REGION Network 1: HS01 / HS02: Contador de veces pulsado sin abrir puerta
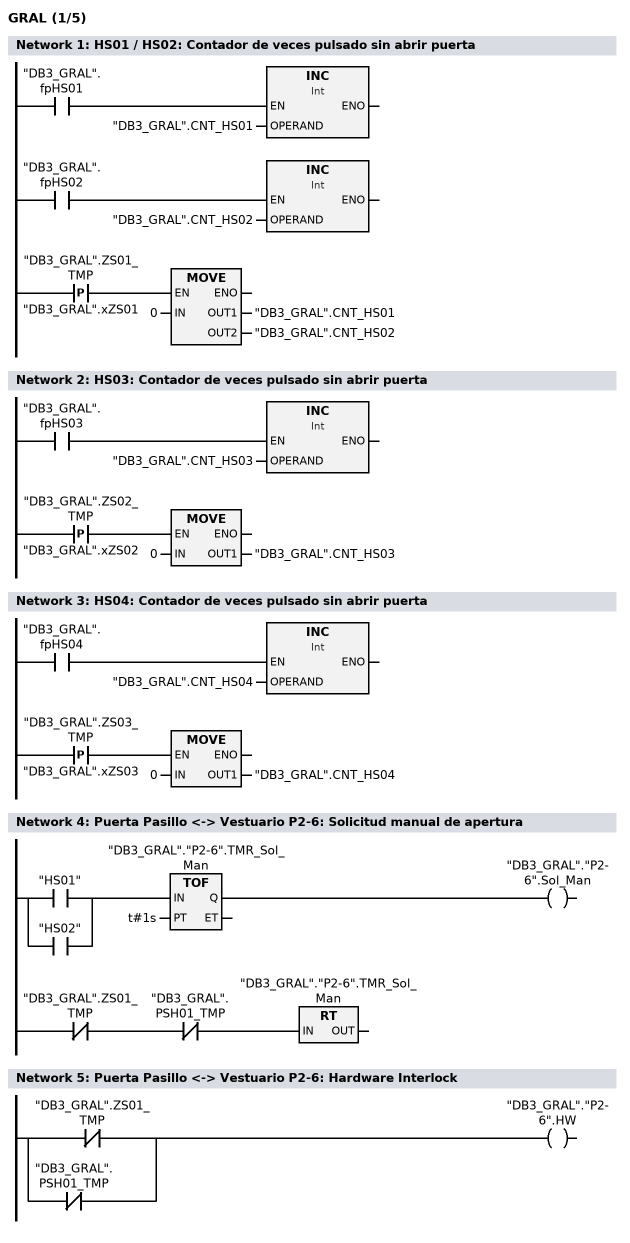
   RUNG wire#powerrail
      Contact( "DB3_GRAL".fpHS01 )
      { S7_Templates := "DestType := Int" } Inc( "DB3_GRAL".CNT_HS01 )
   END_RUNG
   RUNG wire#powerrail
      Contact( "DB3_GRAL".fpHS02 )
      { S7_Templates := "DestType := Int" } Inc( "DB3_GRAL".CNT_HS02 )
   END_RUNG
   RUNG wire#powerrail
      P_Contact(operand := "DB3_GRAL".ZS01_TMP, bit := "DB3_GRAL".xZS01)
      Move(in := 0, out1 => "DB3_GRAL".CNT_HS01, out2 => "DB3_GRAL".CNT_HS02)
   END_RUNG
   // the same network as SCL:
   IF "DB3_GRAL".fpHS01 THEN "DB3_GRAL".CNT_HS01 := "DB3_GRAL".CNT_HS01 + 1; END_IF;
   IF "DB3_GRAL".fpHS02 THEN "DB3_GRAL".CNT_HS02 := "DB3_GRAL".CNT_HS02 + 1; END_IF;
   #_w1 := "DB3_GRAL".ZS01_TMP AND NOT "DB3_GRAL".xZS01;   // rising edge of "DB3_GRAL".ZS01_TMP
   "DB3_GRAL".xZS01 := "DB3_GRAL".ZS01_TMP;
   IF #_w1 THEN
       "DB3_GRAL".CNT_HS01 := 0;
       "DB3_GRAL".CNT_HS02 := 0;
   END_IF;
END_REGION

REGION Network 2: HS03: Contador de veces pulsado sin abrir puerta
   RUNG wire#powerrail
      Contact( "DB3_GRAL".fpHS03 )
      { S7_Templates := "DestType := Int" } Inc( "DB3_GRAL".CNT_HS03 )
   END_RUNG
   RUNG wire#powerrail
      P_Contact(operand := "DB3_GRAL".ZS02_TMP, bit := "DB3_GRAL".xZS02)
      Move(in := 0, out1 => "DB3_GRAL".CNT_HS03)
   END_RUNG
   // the same network as SCL:
   IF "DB3_GRAL".fpHS03 THEN "DB3_GRAL".CNT_HS03 := "DB3_GRAL".CNT_HS03 + 1; END_IF;
   #_w1 := "DB3_GRAL".ZS02_TMP AND NOT "DB3_GRAL".xZS02;   // rising edge of "DB3_GRAL".ZS02_TMP
   "DB3_GRAL".xZS02 := "DB3_GRAL".ZS02_TMP;
   IF #_w1 THEN "DB3_GRAL".CNT_HS03 := 0; END_IF;
END_REGION

REGION Network 3: HS04: Contador de veces pulsado sin abrir puerta
   RUNG wire#powerrail
      Contact( "DB3_GRAL".fpHS04 )
      { S7_Templates := "DestType := Int" } Inc( "DB3_GRAL".CNT_HS04 )
   END_RUNG
   RUNG wire#powerrail
      P_Contact(operand := "DB3_GRAL".ZS03_TMP, bit := "DB3_GRAL".xZS03)
      Move(in := 0, out1 => "DB3_GRAL".CNT_HS04)
   END_RUNG
   // the same network as SCL:
   IF "DB3_GRAL".fpHS04 THEN "DB3_GRAL".CNT_HS04 := "DB3_GRAL".CNT_HS04 + 1; END_IF;
   #_w1 := "DB3_GRAL".ZS03_TMP AND NOT "DB3_GRAL".xZS03;   // rising edge of "DB3_GRAL".ZS03_TMP
   "DB3_GRAL".xZS03 := "DB3_GRAL".ZS03_TMP;
   IF #_w1 THEN "DB3_GRAL".CNT_HS04 := 0; END_IF;
END_REGION

REGION Network 4: Puerta Pasillo <-> Vestuario P2-6: Solicitud manual de apertura
   "DB3_GRAL"."P2-6".TMR_Sol_Man.TOF(IN := "HS01" OR "HS02", PT := t#1s);
   "DB3_GRAL"."P2-6".Sol_Man := "DB3_GRAL"."P2-6".TMR_Sol_Man.Q;
   IF NOT "DB3_GRAL".ZS01_TMP AND NOT "DB3_GRAL".PSH01_TMP THEN
       RESET_TIMER("DB3_GRAL"."P2-6".TMR_Sol_Man);
   END_IF;
END_REGION

REGION Network 5: Puerta Pasillo <-> Vestuario P2-6: Hardware Interlock
   RUNG wire#powerrail
      I_Contact( "DB3_GRAL".ZS01_TMP )
      wire#w1
      Coil( "DB3_GRAL"."P2-6".HW )
   END_RUNG
   RUNG wire#powerrail
      I_Contact( "DB3_GRAL".PSH01_TMP )
   END_RUNG wire#w1
   // the same network as SCL:
   "DB3_GRAL"."P2-6".HW := NOT "DB3_GRAL".ZS01_TMP OR NOT "DB3_GRAL".PSH01_TMP;
END_REGION

REGION Network 6: Puerta Pasillo <-> Vestuario P2-6: Comando apertura
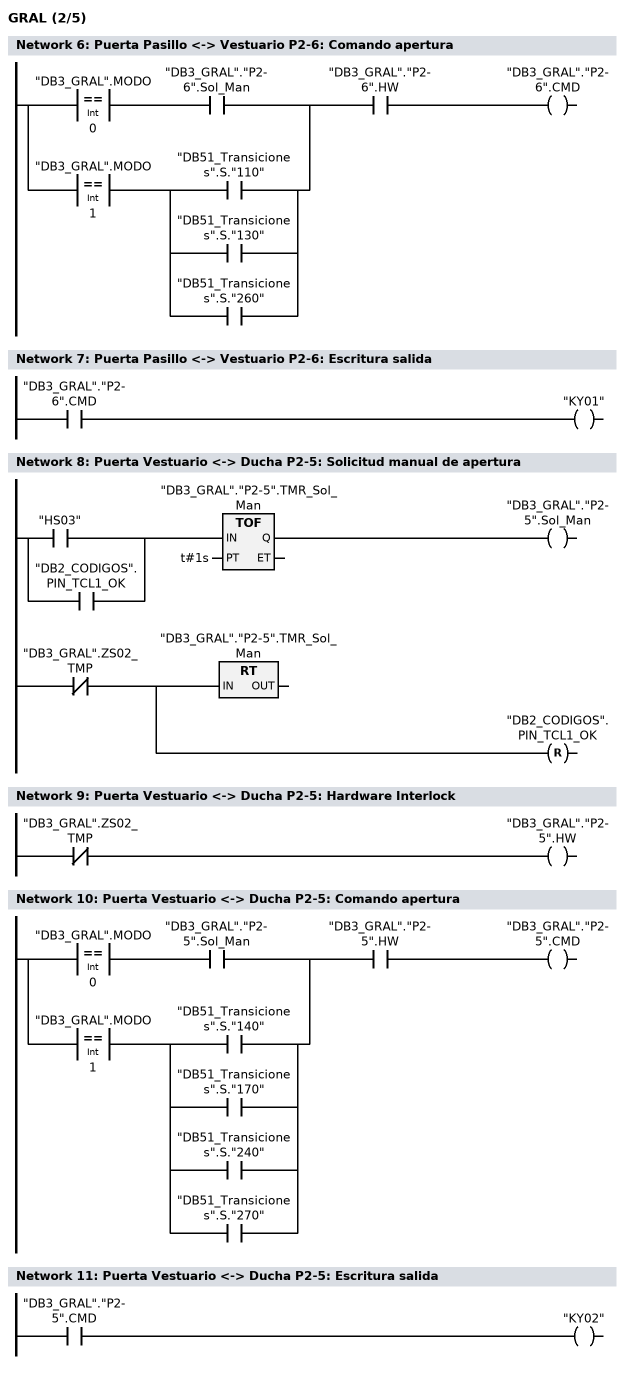
   RUNG wire#powerrail
      { S7_Templates := "SrcType := Int" } EQ_Contact(in1 := "DB3_GRAL".MODO, in2 := 0)
      Contact( "DB3_GRAL"."P2-6".Sol_Man )
      wire#w1
      Contact( "DB3_GRAL"."P2-6".HW )
      Coil( "DB3_GRAL"."P2-6".CMD )
   END_RUNG
   RUNG wire#powerrail
      { S7_Templates := "SrcType := Int" } EQ_Contact(in1 := "DB3_GRAL".MODO, in2 := 1)
      wire#w2
      Contact( "DB51_Transiciones".S."110" )
   END_RUNG wire#w1
   RUNG wire#w2
      Contact( "DB51_Transiciones".S."130" )
   END_RUNG wire#w1
   RUNG wire#w2
      Contact( "DB51_Transiciones".S."260" )
   END_RUNG wire#w1
   // the same network as SCL:
   "DB3_GRAL"."P2-6".CMD := ((("DB3_GRAL".MODO = 0) AND "DB3_GRAL"."P2-6".Sol_Man) OR (("DB3_GRAL".MODO = 1) AND ("DB51_Transiciones".S."110" OR "DB51_Transiciones".S."130" OR "DB51_Transiciones".S."260"))) AND "DB3_GRAL"."P2-6".HW;
END_REGION

REGION Network 7: Puerta Pasillo <-> Vestuario P2-6: Escritura salida
   RUNG wire#powerrail
      Contact( "DB3_GRAL"."P2-6".CMD )
      Coil( "KY01" )
   END_RUNG
   // the same network as SCL:
   "KY01" := "DB3_GRAL"."P2-6".CMD;
END_REGION

REGION Network 8: Puerta Vestuario <-> Ducha P2-5: Solicitud manual de apertura
   "DB3_GRAL"."P2-5".TMR_Sol_Man.TOF(IN := "HS03" OR "DB2_CODIGOS".PIN_TCL1_OK, PT := t#1s);
   "DB3_GRAL"."P2-5".Sol_Man := "DB3_GRAL"."P2-5".TMR_Sol_Man.Q;
   IF NOT "DB3_GRAL".ZS02_TMP THEN
       RESET_TIMER("DB3_GRAL"."P2-5".TMR_Sol_Man);
       "DB2_CODIGOS".PIN_TCL1_OK := FALSE;
   END_IF;
END_REGION

REGION Network 9: Puerta Vestuario <-> Ducha P2-5: Hardware Interlock
   RUNG wire#powerrail
      I_Contact( "DB3_GRAL".ZS02_TMP )
      Coil( "DB3_GRAL"."P2-5".HW )
   END_RUNG
   // the same network as SCL:
   "DB3_GRAL"."P2-5".HW := NOT "DB3_GRAL".ZS02_TMP;
END_REGION

REGION Network 10: Puerta Vestuario <-> Ducha P2-5: Comando apertura
   RUNG wire#powerrail
      { S7_Templates := "SrcType := Int" } EQ_Contact(in1 := "DB3_GRAL".MODO, in2 := 0)
      Contact( "DB3_GRAL"."P2-5".Sol_Man )
      wire#w1
      Contact( "DB3_GRAL"."P2-5".HW )
      Coil( "DB3_GRAL"."P2-5".CMD )
   END_RUNG
   RUNG wire#powerrail
      { S7_Templates := "SrcType := Int" } EQ_Contact(in1 := "DB3_GRAL".MODO, in2 := 1)
      wire#w2
      Contact( "DB51_Transiciones".S."140" )
   END_RUNG wire#w1
   RUNG wire#w2
      Contact( "DB51_Transiciones".S."170" )
   END_RUNG wire#w1
   RUNG wire#w2
      Contact( "DB51_Transiciones".S."240" )
   END_RUNG wire#w1
   RUNG wire#w2
      Contact( "DB51_Transiciones".S."270" )
   END_RUNG wire#w1
   // the same network as SCL:
   "DB3_GRAL"."P2-5".CMD := ((("DB3_GRAL".MODO = 0) AND "DB3_GRAL"."P2-5".Sol_Man) OR (("DB3_GRAL".MODO = 1) AND ("DB51_Transiciones".S."140" OR "DB51_Transiciones".S."170" OR "DB51_Transiciones".S."240" OR "DB51_Transiciones".S."270"))) AND "DB3_GRAL"."P2-5".HW;
END_REGION

REGION Network 11: Puerta Vestuario <-> Ducha P2-5: Escritura salida
   RUNG wire#powerrail
      Contact( "DB3_GRAL"."P2-5".CMD )
      Coil( "KY02" )
   END_RUNG
   // the same network as SCL:
   "KY02" := "DB3_GRAL"."P2-5".CMD;
END_REGION

REGION Network 12: Puerta Ducha <-> Bioterio P2-4: Solicitud manual de apertura
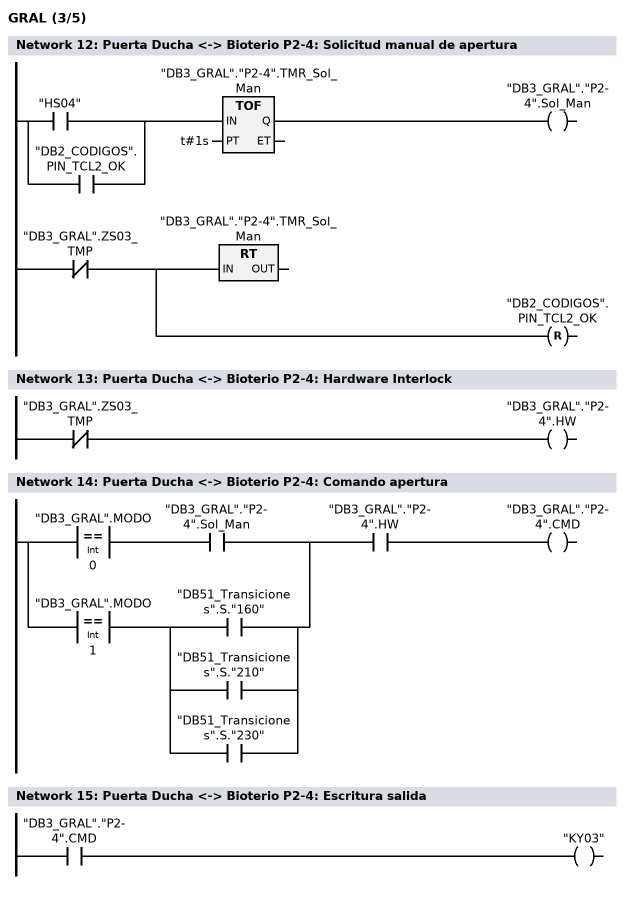
   "DB3_GRAL"."P2-4".TMR_Sol_Man.TOF(IN := "HS04" OR "DB2_CODIGOS".PIN_TCL2_OK, PT := t#1s);
   "DB3_GRAL"."P2-4".Sol_Man := "DB3_GRAL"."P2-4".TMR_Sol_Man.Q;
   IF NOT "DB3_GRAL".ZS03_TMP THEN
       RESET_TIMER("DB3_GRAL"."P2-4".TMR_Sol_Man);
       "DB2_CODIGOS".PIN_TCL2_OK := FALSE;
   END_IF;
END_REGION

REGION Network 13: Puerta Ducha <-> Bioterio P2-4: Hardware Interlock
   RUNG wire#powerrail
      I_Contact( "DB3_GRAL".ZS03_TMP )
      Coil( "DB3_GRAL"."P2-4".HW )
   END_RUNG
   // the same network as SCL:
   "DB3_GRAL"."P2-4".HW := NOT "DB3_GRAL".ZS03_TMP;
END_REGION

REGION Network 14: Puerta Ducha <-> Bioterio P2-4: Comando apertura
   RUNG wire#powerrail
      { S7_Templates := "SrcType := Int" } EQ_Contact(in1 := "DB3_GRAL".MODO, in2 := 0)
      Contact( "DB3_GRAL"."P2-4".Sol_Man )
      wire#w1
      Contact( "DB3_GRAL"."P2-4".HW )
      Coil( "DB3_GRAL"."P2-4".CMD )
   END_RUNG
   RUNG wire#powerrail
      { S7_Templates := "SrcType := Int" } EQ_Contact(in1 := "DB3_GRAL".MODO, in2 := 1)
      wire#w2
      Contact( "DB51_Transiciones".S."160" )
   END_RUNG wire#w1
   RUNG wire#w2
      Contact( "DB51_Transiciones".S."210" )
   END_RUNG wire#w1
   RUNG wire#w2
      Contact( "DB51_Transiciones".S."230" )
   END_RUNG wire#w1
   // the same network as SCL:
   "DB3_GRAL"."P2-4".CMD := ((("DB3_GRAL".MODO = 0) AND "DB3_GRAL"."P2-4".Sol_Man) OR (("DB3_GRAL".MODO = 1) AND ("DB51_Transiciones".S."160" OR "DB51_Transiciones".S."210" OR "DB51_Transiciones".S."230"))) AND "DB3_GRAL"."P2-4".HW;
END_REGION

REGION Network 15: Puerta Ducha <-> Bioterio P2-4: Escritura salida
   RUNG wire#powerrail
      Contact( "DB3_GRAL"."P2-4".CMD )
      Coil( "KY03" )
   END_RUNG
   // the same network as SCL:
   "KY03" := "DB3_GRAL"."P2-4".CMD;
END_REGION

REGION Network 16: Ducha - Electroválvula: Solicitud manual de apertura
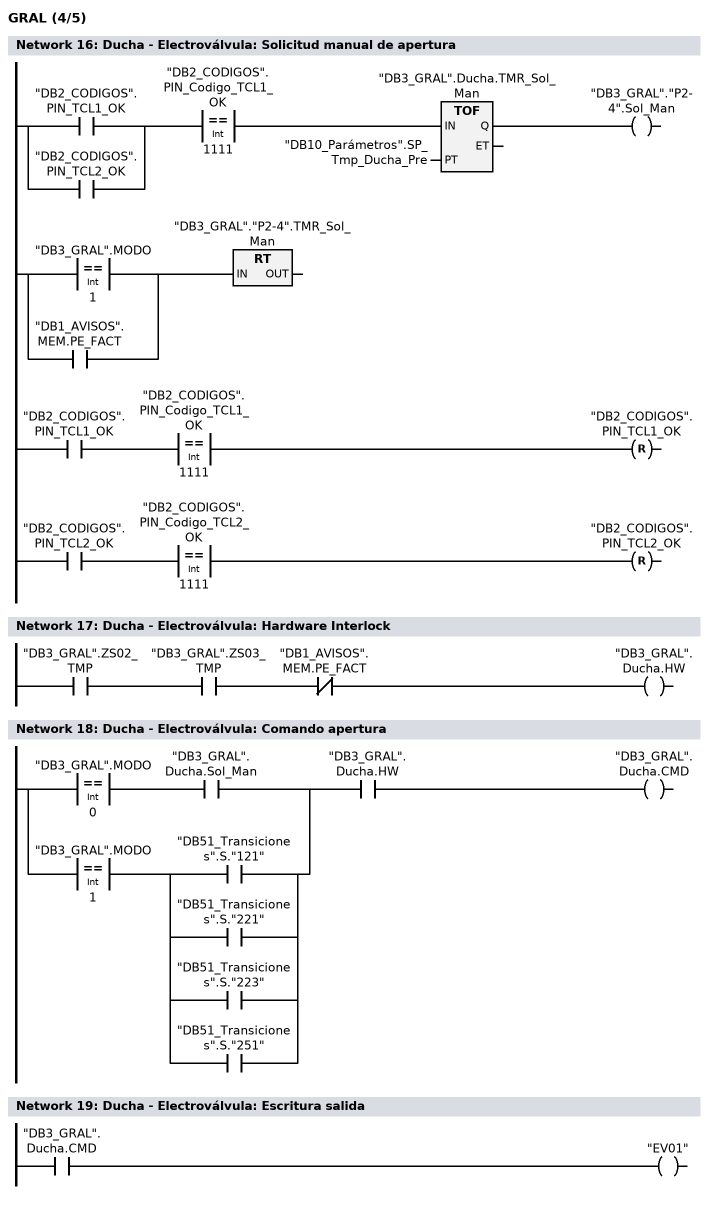
   "DB3_GRAL".Ducha.TMR_Sol_Man.TOF(IN := ("DB2_CODIGOS".PIN_TCL1_OK OR "DB2_CODIGOS".PIN_TCL2_OK) AND ("DB2_CODIGOS".PIN_Codigo_TCL1_OK = 1111),
                           PT := "DB10_Parámetros".SP_Tmp_Ducha_Pre);
   "DB3_GRAL"."P2-4".Sol_Man := "DB3_GRAL".Ducha.TMR_Sol_Man.Q;
   IF ("DB3_GRAL".MODO = 1) OR "DB1_AVISOS".MEM.PE_FACT THEN
       RESET_TIMER("DB3_GRAL"."P2-4".TMR_Sol_Man);
   END_IF;
   IF "DB2_CODIGOS".PIN_TCL1_OK AND ("DB2_CODIGOS".PIN_Codigo_TCL1_OK = 1111) THEN
       "DB2_CODIGOS".PIN_TCL1_OK := FALSE;
   END_IF;
   IF "DB2_CODIGOS".PIN_TCL2_OK AND ("DB2_CODIGOS".PIN_Codigo_TCL2_OK = 1111) THEN
       "DB2_CODIGOS".PIN_TCL2_OK := FALSE;
   END_IF;
END_REGION

REGION Network 17: Ducha - Electroválvula: Hardware Interlock
   RUNG wire#powerrail
      Contact( "DB3_GRAL".ZS02_TMP )
      Contact( "DB3_GRAL".ZS03_TMP )
      I_Contact( "DB1_AVISOS".MEM.PE_FACT )
      Coil( "DB3_GRAL".Ducha.HW )
   END_RUNG
   // the same network as SCL:
   "DB3_GRAL".Ducha.HW := "DB3_GRAL".ZS02_TMP AND "DB3_GRAL".ZS03_TMP AND NOT "DB1_AVISOS".MEM.PE_FACT;
END_REGION

REGION Network 18: Ducha - Electroválvula: Comando apertura
   RUNG wire#powerrail
      { S7_Templates := "SrcType := Int" } EQ_Contact(in1 := "DB3_GRAL".MODO, in2 := 0)
      Contact( "DB3_GRAL".Ducha.Sol_Man )
      wire#w1
      Contact( "DB3_GRAL".Ducha.HW )
      Coil( "DB3_GRAL".Ducha.CMD )
   END_RUNG
   RUNG wire#powerrail
      { S7_Templates := "SrcType := Int" } EQ_Contact(in1 := "DB3_GRAL".MODO, in2 := 1)
      wire#w2
      Contact( "DB51_Transiciones".S."121" )
   END_RUNG wire#w1
   RUNG wire#w2
      Contact( "DB51_Transiciones".S."221" )
   END_RUNG wire#w1
   RUNG wire#w2
      Contact( "DB51_Transiciones".S."223" )
   END_RUNG wire#w1
   RUNG wire#w2
      Contact( "DB51_Transiciones".S."251" )
   END_RUNG wire#w1
   // the same network as SCL:
   "DB3_GRAL".Ducha.CMD := ((("DB3_GRAL".MODO = 0) AND "DB3_GRAL".Ducha.Sol_Man) OR (("DB3_GRAL".MODO = 1) AND ("DB51_Transiciones".S."121" OR "DB51_Transiciones".S."221" OR "DB51_Transiciones".S."223" OR "DB51_Transiciones".S."251"))) AND "DB3_GRAL".Ducha.HW;
END_REGION

REGION Network 19: Ducha - Electroválvula: Escritura salida
   RUNG wire#powerrail
      Contact( "DB3_GRAL".Ducha.CMD )
      Coil( "EV01" )
   END_RUNG
   // the same network as SCL:
   "EV01" := "DB3_GRAL".Ducha.CMD;
END_REGION

REGION Network 20: *****************************************************
END_REGION

REGION Network 21: Contador de personas que ingresaron al bioterio
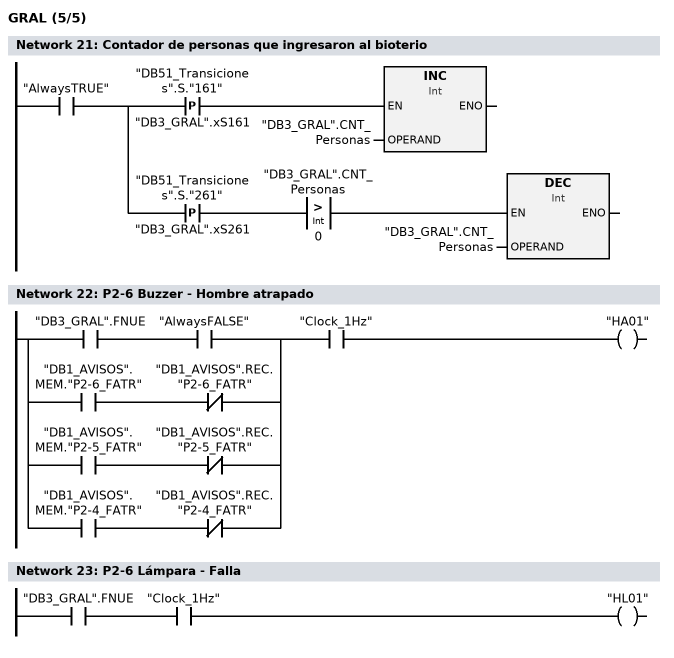
   RUNG wire#powerrail
      Contact( "AlwaysTRUE" )
      wire#w1
      P_Contact(operand := "DB51_Transiciones".S."161", bit := "DB3_GRAL".xS161)
      { S7_Templates := "DestType := Int" } Inc( "DB3_GRAL".CNT_Personas )
   END_RUNG
   RUNG wire#w1
      P_Contact(operand := "DB51_Transiciones".S."261", bit := "DB3_GRAL".xS261)
      { S7_Templates := "SrcType := Int" } GT_Contact(in1 := "DB3_GRAL".CNT_Personas, in2 := 0)
      { S7_Templates := "DestType := Int" } Dec( "DB3_GRAL".CNT_Personas )
   END_RUNG
   // the same network as SCL:
   #_w1 := "AlwaysTRUE" AND "DB51_Transiciones".S."161" AND NOT "DB3_GRAL".xS161;   // rising edge of "DB51_Transiciones".S."161"
   "DB3_GRAL".xS161 := "DB51_Transiciones".S."161";
   IF #_w1 THEN "DB3_GRAL".CNT_Personas := "DB3_GRAL".CNT_Personas + 1; END_IF;
   #_w2 := "AlwaysTRUE" AND "DB51_Transiciones".S."261" AND NOT "DB3_GRAL".xS261;   // rising edge of "DB51_Transiciones".S."261"
   "DB3_GRAL".xS261 := "DB51_Transiciones".S."261";
   IF #_w2 AND ("DB3_GRAL".CNT_Personas > 0) THEN
       "DB3_GRAL".CNT_Personas := "DB3_GRAL".CNT_Personas - 1;
   END_IF;
END_REGION

REGION Network 22: P2-6 Buzzer - Hombre atrapado
   RUNG wire#powerrail
      Contact( "DB3_GRAL".FNUE )
      Contact( "AlwaysFALSE" )
      wire#w1
      Contact( "Clock_1Hz" )
      Coil( "HA01" )
   END_RUNG
   RUNG wire#powerrail
      Contact( "DB1_AVISOS".MEM."P2-6_FATR" )
      I_Contact( "DB1_AVISOS".REC."P2-6_FATR" )
   END_RUNG wire#w1
   RUNG wire#powerrail
      Contact( "DB1_AVISOS".MEM."P2-5_FATR" )
      I_Contact( "DB1_AVISOS".REC."P2-5_FATR" )
   END_RUNG wire#w1
   RUNG wire#powerrail
      Contact( "DB1_AVISOS".MEM."P2-4_FATR" )
      I_Contact( "DB1_AVISOS".REC."P2-4_FATR" )
   END_RUNG wire#w1
   // the same network as SCL:
   "HA01" := (("DB3_GRAL".FNUE AND "AlwaysFALSE") OR ("DB1_AVISOS".MEM."P2-6_FATR" AND NOT "DB1_AVISOS".REC."P2-6_FATR") OR ("DB1_AVISOS".MEM."P2-5_FATR" AND NOT "DB1_AVISOS".REC."P2-5_FATR") OR ("DB1_AVISOS".MEM."P2-4_FATR" AND NOT "DB1_AVISOS".REC."P2-4_FATR")) AND "Clock_1Hz";
END_REGION

REGION Network 23: P2-6 Lámpara - Falla
   RUNG wire#powerrail
      Contact( "DB3_GRAL".FNUE )
      Contact( "Clock_1Hz" )
      Coil( "HL01" )
   END_RUNG
   // the same network as SCL:
   "HL01" := "DB3_GRAL".FNUE AND "Clock_1Hz";
END_REGION
END_FUNCTION

FUNCTION "INICIA" : Void   // FC5, LAD
TITLE = Inicialización de datos
{ S7_Optimized_Access := 'TRUE' }
AUTHOR : IGLP
VERSION : 0.1
BEGIN

REGION Network 1: Contacto Magnético P2-6 - Temporizado
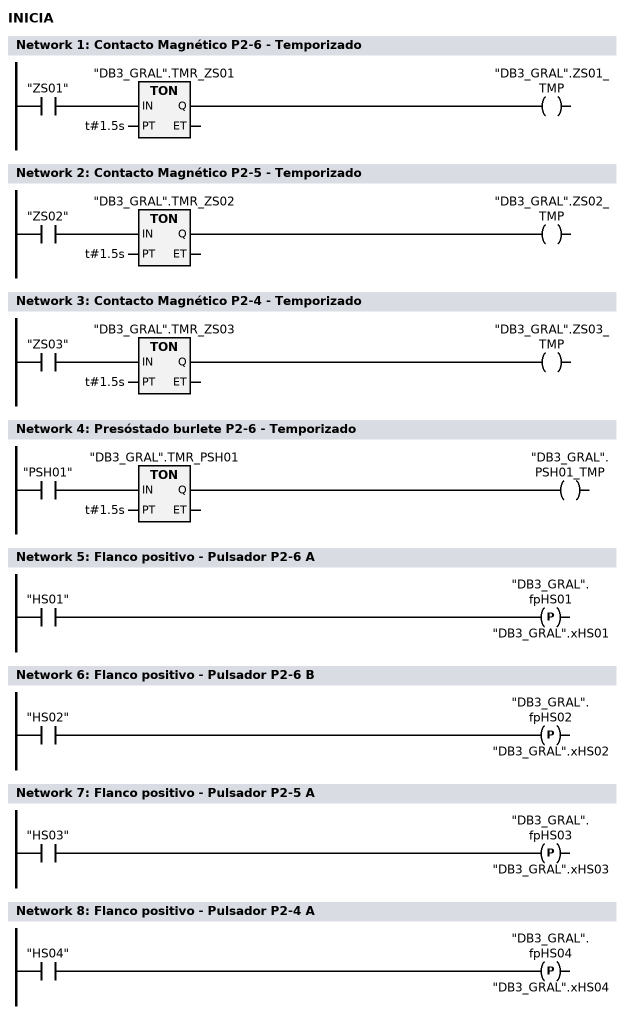
   "DB3_GRAL".TMR_ZS01.TON(IN := "ZS01", PT := t#1.5s);
   "DB3_GRAL".ZS01_TMP := "DB3_GRAL".TMR_ZS01.Q;
END_REGION

REGION Network 2: Contacto Magnético P2-5 - Temporizado
   "DB3_GRAL".TMR_ZS02.TON(IN := "ZS02", PT := t#1.5s);
   "DB3_GRAL".ZS02_TMP := "DB3_GRAL".TMR_ZS02.Q;
END_REGION

REGION Network 3: Contacto Magnético P2-4 - Temporizado
   "DB3_GRAL".TMR_ZS03.TON(IN := "ZS03", PT := t#1.5s);
   "DB3_GRAL".ZS03_TMP := "DB3_GRAL".TMR_ZS03.Q;
END_REGION

REGION Network 4: Presóstado burlete P2-6 - Temporizado
   "DB3_GRAL".TMR_PSH01.TON(IN := "PSH01", PT := t#1.5s);
   "DB3_GRAL".PSH01_TMP := "DB3_GRAL".TMR_PSH01.Q;
END_REGION

REGION Network 5: Flanco positivo - Pulsador P2-6 A
   "DB3_GRAL".fpHS01 := "HS01" AND NOT "DB3_GRAL".xHS01;   // rising edge
   "DB3_GRAL".xHS01 := "HS01";
END_REGION

REGION Network 6: Flanco positivo - Pulsador P2-6 B
   "DB3_GRAL".fpHS02 := "HS02" AND NOT "DB3_GRAL".xHS02;   // rising edge
   "DB3_GRAL".xHS02 := "HS02";
END_REGION

REGION Network 7: Flanco positivo - Pulsador P2-5 A
   "DB3_GRAL".fpHS03 := "HS03" AND NOT "DB3_GRAL".xHS03;   // rising edge
   "DB3_GRAL".xHS03 := "HS03";
END_REGION

REGION Network 8: Flanco positivo - Pulsador P2-4 A
   "DB3_GRAL".fpHS04 := "HS04" AND NOT "DB3_GRAL".xHS04;   // rising edge
   "DB3_GRAL".xHS04 := "HS04";
END_REGION
END_FUNCTION

FUNCTION "AVISOS" : Void   // FC6, LAD
TITLE = Avisos
{ S7_Optimized_Access := 'TRUE' }
AUTHOR : IGLP
VERSION : 0.1
BEGIN

REGION Network 1: Falla: Emergencia actuada
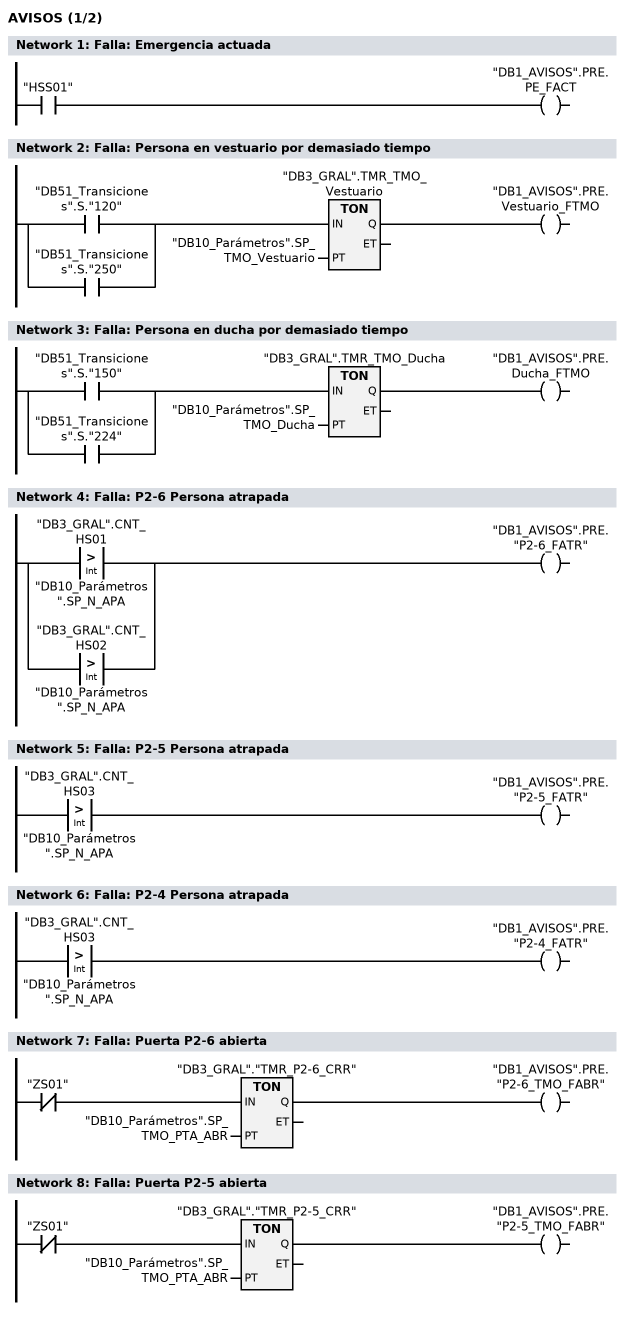
   RUNG wire#powerrail
      Contact( "HSS01" )
      Coil( "DB1_AVISOS".PRE.PE_FACT )
   END_RUNG
   // the same network as SCL:
   "DB1_AVISOS".PRE.PE_FACT := "HSS01";
END_REGION

REGION Network 2: Falla: Persona en vestuario por demasiado tiempo
   "DB3_GRAL".TMR_TMO_Vestuario.TON(IN := "DB51_Transiciones".S."120" OR "DB51_Transiciones".S."250",
                           PT := "DB10_Parámetros".SP_TMO_Vestuario);
   "DB1_AVISOS".PRE.Vestuario_FTMO := "DB3_GRAL".TMR_TMO_Vestuario.Q;
END_REGION

REGION Network 3: Falla: Persona en ducha por demasiado tiempo
   "DB3_GRAL".TMR_TMO_Ducha.TON(IN := "DB51_Transiciones".S."150" OR "DB51_Transiciones".S."224",
                           PT := "DB10_Parámetros".SP_TMO_Ducha);
   "DB1_AVISOS".PRE.Ducha_FTMO := "DB3_GRAL".TMR_TMO_Ducha.Q;
END_REGION

REGION Network 4: Falla: P2-6 Persona atrapada
   RUNG wire#powerrail
      { S7_Templates := "SrcType := Int" } GT_Contact(in1 := "DB3_GRAL".CNT_HS01, in2 := "DB10_Parámetros".SP_N_APA)
      wire#w1
      Coil( "DB1_AVISOS".PRE."P2-6_FATR" )
   END_RUNG
   RUNG wire#powerrail
      { S7_Templates := "SrcType := Int" } GT_Contact(in1 := "DB3_GRAL".CNT_HS02, in2 := "DB10_Parámetros".SP_N_APA)
   END_RUNG wire#w1
   // the same network as SCL:
   "DB1_AVISOS".PRE."P2-6_FATR" := ("DB3_GRAL".CNT_HS01 > "DB10_Parámetros".SP_N_APA) OR ("DB3_GRAL".CNT_HS02 > "DB10_Parámetros".SP_N_APA);
END_REGION

REGION Network 5: Falla: P2-5 Persona atrapada
   RUNG wire#powerrail
      { S7_Templates := "SrcType := Int" } GT_Contact(in1 := "DB3_GRAL".CNT_HS03, in2 := "DB10_Parámetros".SP_N_APA)
      Coil( "DB1_AVISOS".PRE."P2-5_FATR" )
   END_RUNG
   // the same network as SCL:
   "DB1_AVISOS".PRE."P2-5_FATR" := "DB3_GRAL".CNT_HS03 > "DB10_Parámetros".SP_N_APA;
END_REGION

REGION Network 6: Falla: P2-4 Persona atrapada
   RUNG wire#powerrail
      { S7_Templates := "SrcType := Int" } GT_Contact(in1 := "DB3_GRAL".CNT_HS03, in2 := "DB10_Parámetros".SP_N_APA)
      Coil( "DB1_AVISOS".PRE."P2-4_FATR" )
   END_RUNG
   // the same network as SCL:
   "DB1_AVISOS".PRE."P2-4_FATR" := "DB3_GRAL".CNT_HS03 > "DB10_Parámetros".SP_N_APA;
END_REGION

REGION Network 7: Falla: Puerta P2-6 abierta
   "DB3_GRAL"."TMR_P2-6_CRR".TON(IN := NOT "ZS01", PT := "DB10_Parámetros".SP_TMO_PTA_ABR);
   "DB1_AVISOS".PRE."P2-6_TMO_FABR" := "DB3_GRAL"."TMR_P2-6_CRR".Q;
END_REGION

REGION Network 8: Falla: Puerta P2-5 abierta
   "DB3_GRAL"."TMR_P2-5_CRR".TON(IN := NOT "ZS01", PT := "DB10_Parámetros".SP_TMO_PTA_ABR);
   "DB1_AVISOS".PRE."P2-5_TMO_FABR" := "DB3_GRAL"."TMR_P2-5_CRR".Q;
END_REGION

REGION Network 9: Falla: Puerta P2-4 abierta
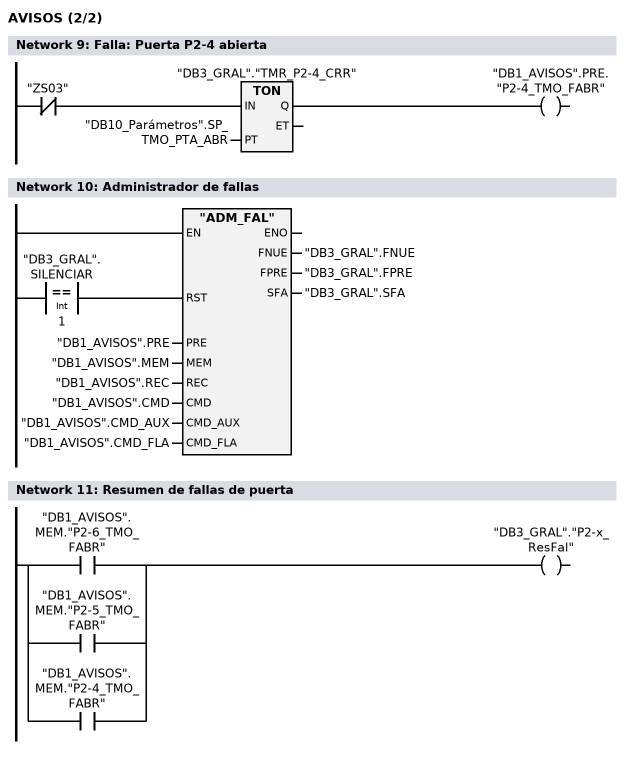
   "DB3_GRAL"."TMR_P2-4_CRR".TON(IN := NOT "ZS03", PT := "DB10_Parámetros".SP_TMO_PTA_ABR);
   "DB1_AVISOS".PRE."P2-4_TMO_FABR" := "DB3_GRAL"."TMR_P2-4_CRR".Q;
END_REGION

REGION Network 10: Administrador de fallas
   RUNG wire#powerrail
      "ADM_FAL"(RST := wire#w1, PRE := "DB1_AVISOS".PRE, MEM := "DB1_AVISOS".MEM, REC := "DB1_AVISOS".REC, CMD := "DB1_AVISOS".CMD, CMD_AUX := "DB1_AVISOS".CMD_AUX, CMD_FLA := "DB1_AVISOS".CMD_FLA, FNUE => "DB3_GRAL".FNUE, FPRE => "DB3_GRAL".FPRE, SFA => "DB3_GRAL".SFA)
   END_RUNG
   RUNG wire#powerrail
      { S7_Templates := "SrcType := Int" } EQ_Contact(in1 := "DB3_GRAL".SILENCIAR, in2 := 1)
   END_RUNG wire#w1
   // the same network as SCL:
   "ADM_FAL"(RST := "DB3_GRAL".SILENCIAR = 1,
             PRE := "DB1_AVISOS".PRE,
             MEM := "DB1_AVISOS".MEM,
             REC := "DB1_AVISOS".REC,
             CMD := "DB1_AVISOS".CMD,
             CMD_AUX := "DB1_AVISOS".CMD_AUX,
             CMD_FLA := "DB1_AVISOS".CMD_FLA,
             FNUE => "DB3_GRAL".FNUE,
             FPRE => "DB3_GRAL".FPRE,
             SFA => "DB3_GRAL".SFA);
END_REGION

REGION Network 11: Resumen de fallas de puerta
   RUNG wire#powerrail
      Contact( "DB1_AVISOS".MEM."P2-6_TMO_FABR" )
      wire#w1
      Coil( "DB3_GRAL"."P2-x_ResFal" )
   END_RUNG
   RUNG wire#powerrail
      Contact( "DB1_AVISOS".MEM."P2-5_TMO_FABR" )
   END_RUNG wire#w1
   RUNG wire#powerrail
      Contact( "DB1_AVISOS".MEM."P2-4_TMO_FABR" )
   END_RUNG wire#w1
   // the same network as SCL:
   "DB3_GRAL"."P2-x_ResFal" := "DB1_AVISOS".MEM."P2-6_TMO_FABR" OR "DB1_AVISOS".MEM."P2-5_TMO_FABR" OR "DB1_AVISOS".MEM."P2-4_TMO_FABR";
END_REGION
END_FUNCTION

FUNCTION "ADM_FAL" : Void   // FC7, LAD
TITLE = Procesador de fallas
{ S7_Optimized_Access := 'FALSE' }
VERSION : 0.1
   VAR_INPUT
      RST : Bool;
   END_VAR
   VAR_OUTPUT
      FNUE : Bool;
      FPRE : Bool;
      SFA : Bool;
   END_VAR
   VAR_IN_OUT
      PRE : "FALLAS";
      aPRE AT PRE : Array[1..2] of Byte;
      MEM : "FALLAS";
      aMEM AT MEM : Array[1..2] of Byte;
      REC : "FALLAS";
      aREC AT REC : Array[1..2] of Byte;
      CMD : "FALLAS";
      aCMD AT CMD : Array[1..2] of Byte;
      CMD_AUX : "FALLAS";
      aCMD_AUX AT CMD_AUX : Array[1..2] of Byte;
      CMD_FLA : "FALLAS";
      aCMD_FLA AT CMD_FLA : Array[1..2] of Byte;
   END_VAR
   VAR_TEMP
      INDICE : Int;
      AUX_FLA_CMD_REC : Byte;
      AUX_Reconocida1 : Byte;
      AUX_Reconocida2 : Byte;
   END_VAR
BEGIN

REGION Network 1: Inicializo
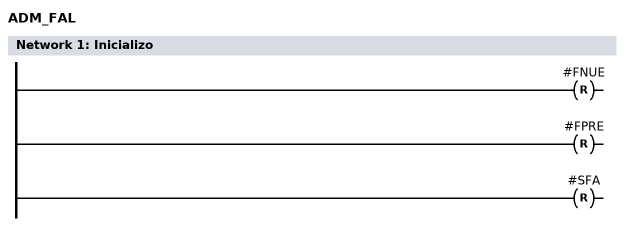
   RUNG wire#powerrail
      R_Coil( #FNUE )
   END_RUNG
   RUNG wire#powerrail
      R_Coil( #FPRE )
   END_RUNG
   RUNG wire#powerrail
      R_Coil( #SFA )
   END_RUNG
   // the same network as SCL:
   #FNUE := FALSE;
   #FPRE := FALSE;
   #SFA := FALSE;
END_REGION

REGION Network 2 (SCL): Comandos reconocimiento: Detección de flancos
   FOR #INDICE := 1 TO 2 DO
       #aCMD_FLA[#INDICE] := (#aCMD[#INDICE] XOR #aCMD_AUX[#INDICE]);
       #aCMD_AUX[#INDICE] := #aCMD[#INDICE];
   END_FOR;
END_REGION

REGION Network 3 (SCL): Memorizo alarmas y reconozco cuando llega flanco
   // Sobre las alarmas reconocidas hay dos operaciones:
   // Set =   (NO(Alarma Presente) * NO(Alarma Memorizada))  + (Alarma Memorizada * Flanco Cmd. Reconocimiento)
   // 
   // Reset= Alarma Presente * NO(Alarma Memorizada)
   // 
   // Notas:
   // 1- El estado normal de una alarma reconocida es "1"
   // 2- La alarma reconocida pasa a "0" con alarma presente
   // 3- Con el flanco del comando de reconocimiento vuelve al estado "1"
   // __________________________________________________________________
   // 
   // Sobre las alarmas memorizadas hay dos operaciones:
   // Set =   Alarma Presente
   // 
   // Reset= NO.Alarma Presente * Alarma Memorizada
   // 
   // Notas:
   // 1- El estado normal de una alarma memorizada es "0"
   // 2- La alarma memorizada pasa a "1" con alarma presente
   // 3- Si no hay alarma reconocida y no hay alarma presente vuelve a "0"
   FOR #INDICE := 1 TO 2 DO
       // Alarmas reconocidas
       IF #RST THEN
           #AUX_FLA_CMD_REC := 16#FF;
       ELSE
           #AUX_FLA_CMD_REC := #aCMD_FLA[#INDICE];
       END_IF;
       #AUX_Reconocida1 := (NOT (#aPRE[#INDICE]) AND NOT (#aMEM[#INDICE])) OR (#aMEM[#INDICE] AND #AUX_FLA_CMD_REC); // Equivale a SET
       #AUX_Reconocida2 := (#aPRE[#INDICE]) AND NOT (#aMEM[#INDICE]); // Equivale a RESET
       #aREC[#INDICE] := #aREC[#INDICE] OR #AUX_Reconocida1;
       #aREC[#INDICE] := #aREC[#INDICE] AND NOT (#AUX_Reconocida2);

       // Alarmas memorizadas
       #aMEM[#INDICE] := #aMEM[#INDICE] OR #aPRE[#INDICE];
       #aMEM[#INDICE] := NOT (NOT (#aPRE[#INDICE]) AND #aREC[#INDICE]);

   END_FOR;
END_REGION

REGION Network 4 (SCL): Reviso si hay alarmas presentes y si hay nuevas
   #SFA := TRUE;
   #FNUE := FALSE;


   FOR #INDICE := 1 TO 2 DO
       IF #aMEM[#INDICE] <> W#16#0 THEN
           #SFA := FALSE;
       END_IF;

       IF (#aMEM[#INDICE] AND NOT #aREC[#INDICE]) <> W#16#0 THEN
           #FNUE := true;
       END_IF;

       IF NOT #SFA AND #FNUE THEN
           EXIT;
       END_IF;

   END_FOR;
END_REGION

REGION Network 5 (SCL): Hay alarmas y reconocidas
   IF (NOT #SFA AND NOT #FNUE) THEN
       #FPRE := TRUE;
   END_IF;
END_REGION
END_FUNCTION

ORGANIZATION_BLOCK "Main"   // OB1, LAD, ProgramCycle
TITLE = "Main Program Sweep (Cycle)"
{ S7_Optimized_Access := 'TRUE' }
VERSION : 0.1
   VAR_INPUT
      Initial_Call : Bool;   // Initial call of this OB
      Remanence : Bool;   // =True, if remanent data are available
   END_VAR
BEGIN

REGION Network 1: Inicializa
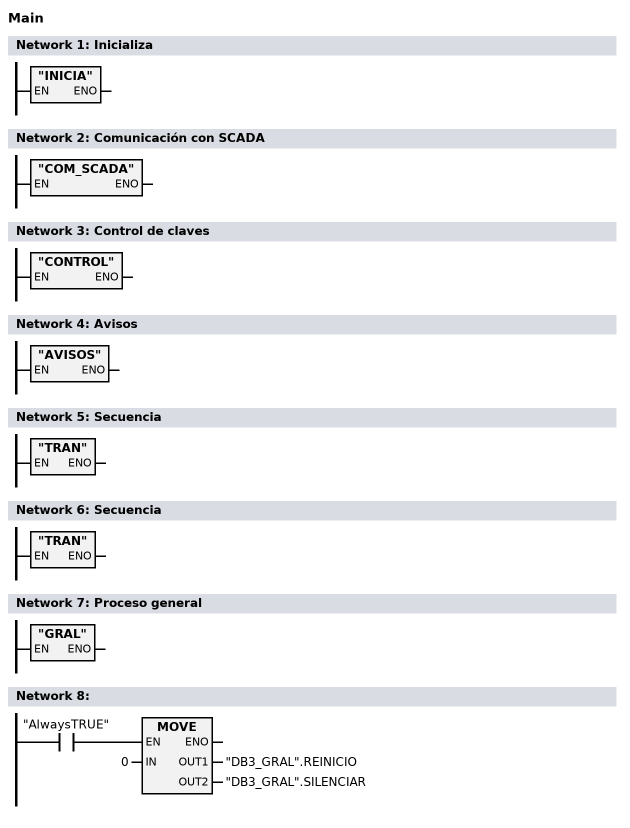
   RUNG wire#powerrail
      "INICIA"()
   END_RUNG
   // the same network as SCL:
   "INICIA"();
END_REGION

REGION Network 2: Comunicación con SCADA
   RUNG wire#powerrail
      "COM_SCADA"()
   END_RUNG
   // the same network as SCL:
   "COM_SCADA"();
END_REGION

REGION Network 3: Control de claves
   RUNG wire#powerrail
      "CONTROL"()
   END_RUNG
   // the same network as SCL:
   "CONTROL"();
END_REGION

REGION Network 4: Avisos
   RUNG wire#powerrail
      "AVISOS"()
   END_RUNG
   // the same network as SCL:
   "AVISOS"();
END_REGION

REGION Network 5: Secuencia
   RUNG wire#powerrail
      "TRAN"()
   END_RUNG
   // the same network as SCL:
   "TRAN"();
END_REGION

REGION Network 6: Secuencia
   RUNG wire#powerrail
      "TRAN"()
   END_RUNG
   // the same network as SCL:
   "TRAN"();
END_REGION

REGION Network 7: Proceso general
   RUNG wire#powerrail
      "GRAL"()
   END_RUNG
   // the same network as SCL:
   "GRAL"();
END_REGION

REGION Network 8
   RUNG wire#powerrail
      Contact( "AlwaysTRUE" )
      Move(in := 0, out1 => "DB3_GRAL".REINICIO, out2 => "DB3_GRAL".SILENCIAR)
   END_RUNG
   // the same network as SCL:
   IF "AlwaysTRUE" THEN
       "DB3_GRAL".REINICIO := 0;
       "DB3_GRAL".SILENCIAR := 0;
   END_IF;
END_REGION
END_ORGANIZATION_BLOCK